// TIA Portal project "CP-AM-DRILL" (V14)

(* hardware
DEVICE "ET 200SP station_1"  ET 200SP-Station
   slot 0: "Rack_0"  Rack  6ES5 710-8MAx1
   slot 1: "PLC_1"  CPU 1512SP F-1 PN  6ES7 512-1SK01-0AB0  V2.1
   slot 2: "DI 8x24VDC HF_1"  DI 8x24VDC HF  6ES7 131-6BF00-0CA0  V2.0
      slot 1: "DI 8x24VDC HF_1"  DI 8x24VDC HF
   slot 3: "DI 8x24VDC HF_2"  DI 8x24VDC HF  6ES7 131-6BF00-0CA0  V2.0
      slot 1: "DI 8x24VDC HF_2"  DI 8x24VDC HF
   slot 4: "DQ 8x24VDC/0.5A HF_1"  DQ 8x24VDC/0.5A HF  6ES7 132-6BF00-0CA0  V2.0
      slot 1: "DQ 8x24VDC/0.5A HF_1"  DQ 8x24VDC/0.5A HF
   slot 5: "DQ 8x24VDC/0.5A HF_2"  DQ 8x24VDC/0.5A HF  6ES7 132-6BF00-0CA0  V2.0
      slot 1: "DQ 8x24VDC/0.5A HF_2"  DQ 8x24VDC/0.5A HF
   slot 6: "Server module_1"  Server module  6ES7 193-6PA00-0AA0  V1.1
      slot 1: "Server module_1"  Server module
   slot 127: "BA 2xRJ45"  BA 2xRJ45  6ES7 193-6AR00-0AA0  V0.0
      slot 32769: "Port_1"  6ES7 193-6AR00-0AA0
      slot 32770: "Port_2"  6ES7 193-6AR00-0AA0
*)

// ===== PLC "PLC_1"  CPU 1512SP F-1 PN =====

VAR_GLOBAL   // PLC tag table "Default tag table"
   "DI1-0" AT %I1.0 : Bool;   // Start button pushed
   "DI1-3" AT %I1.3 : Bool;   // Reset button pushed
   "DI1-6" AT %I1.6 : Bool;   // Carrier detected at conveyor entry
   "DI1-7" AT %I1.7 : Bool;   // Carrier detected at conveyor exit
   "DI18-0" AT %I18.0 : Bool;   // Carrier ident code bit 0 detected
   "DI18-1" AT %I18.1 : Bool;   // Carrier ident code bit 1 detected
   "DI18-2" AT %I18.2 : Bool;   // Carrier ident code bit 2 detected
   "DI18-3" AT %I18.3 : Bool;   // Carrier ident code bit 3 detected
   "DI18-7" AT %I18.7 : Bool;   // Stopper in lower position
   "DQ1-0" AT %Q1.0 : Bool;   // Switch on "start button signal light"
   "DQ1-1" AT %Q1.1 : Bool;   // Switch on "reset button signal light"
   "DQ1-2" AT %Q1.2 : Bool;   // Switch on "special function Q1 signal light"
   "DQ1-3" AT %Q1.3 : Bool;   // Switch on "special function Q2 signal light"
   "DQ1-4" AT %Q1.4 : Bool;   // Drive conveyor belt in forward direction
   "DQ1-5" AT %Q1.5 : Bool;   // Drive conveyor belt in backward direction
   "DQ1-7" AT %Q1.7 : Bool;   // Move stopper downwards
   "DI1-1" AT %I1.1 : Bool;   // Stop button pushed
   "DI0-0" AT %I0.0 : Bool;   // X-axis in left end position
   "DI0-1" AT %I0.1 : Bool;   // X-axis in right end position
   "DI0-2" AT %I0.2 : Bool;   // Front cover orientation NOT correct
   "DI0-3" AT %I0.3 : Bool;   // Front cover present
   "DI0-4" AT %I0.4 : Bool;   // Z-axis in upper end position
   "DI0-5" AT %I0.5 : Bool;   // Z-axis in lower end position
   "DI0-7" AT %I0.7 : Bool;   // Backcover already present
   "DQ0-0" AT %Q0.0 : Bool;   // Move X-axis left
   "DQ0-1" AT %Q0.1 : Bool;   // Move X-axis right
   "DQ0-2" AT %Q0.2 : Bool;   // Switch on drill 1
   "DQ0-3" AT %Q0.3 : Bool;   // Switch on drill 2
   "DQ0-4" AT %Q0.4 : Bool;   // Move Z-axis up
   "DQ0-5" AT %Q0.5 : Bool;   // Move Z-axis down
   "DQ0-6" AT %Q0.6 : Bool;   // Open Z-axis end position lock
END_VAR

ORGANIZATION_BLOCK "Main"   // OB1, LAD, ProgramCycle
TITLE = "Main Program Sweep (Cycle)"
{ S7_Optimized_Access := 'TRUE' }
VERSION : 0.1
   VAR_INPUT
      Initial_Call : Bool;   // Initial call of this OB
      Remanence : Bool;   // =True, if remanent data are available
   END_VAR
BEGIN
END_ORGANIZATION_BLOCK